// Diagnostic marker interface.
INTERFACE I_Debug

END_INTERFACE

(* stored: Version 1.1.0.1
   Itf I_Debug: Id {dd9af94b-653d-4389-8fe6-660d00f8293a} *)
